(* IEC 61131-3 sources: SigmatekTestframework/src/Class/CTestScreen, 1 file *)

(* ---- CTestScreen.st ---- *)
(*!
<Class
	Name               = "CTestScreen"
	Revision           = "1.0"
	RealtimeTask       = "false"
	CyclicTask         = "false"
	BackgroundTask     = "false"
	Sigmatek           = "false"
	OSInterface        = "false"
	HighPriority       = "false"
	Automatic          = "false"
	UpdateMode         = "Prescan"
	IconPath           = ".\Class\CTestScreen\TestIcon36x36.ico"
	SharedCommandTable = "true"
	Objectsize         = "(450,120)"
	Comment            = "Base Class for Lasal Screen Testing">
	<Channels>
		<Client Name="Lse" Required="true" Internal="false" Comment="Connect to _LSE Runtime"/>
		<Client Name="m_Screen" Required="true" Internal="true"/>
		<Client Name="No" Required="true" Internal="false" Comment="Number of Screen from Lasal Screen Project"/>
	</Channels>
	<Network Name="CTestScreen">
		<!-- List of Components in this network -->
		<Components>
			<Object
				Name       = "_base"
				Class      = "CTestBase"
				Position   = "(218,120)"
				Visualized = "true">
				<Channels>
					<Server Name="Deactivate"/>
					<Server Name="State"/>
					<Client Name="cLib"/>
					<Client Name="TestSuite"/>
				</Channels>
			</Object>
			<Object
				Name       = "m_Screen"
				Class      = "CScreenInterface"
				Position   = "(210,480)"
				Visualized = "true"
				Remotely   = "true">
				<Channels>
					<Server Name="Active"/>
					<Server Name="Screen"/>
					<Client Name="ImA" Value="IMA_PICTURE"/>
					<Client Name="Lse"/>
					<Client Name="No"/>
				</Channels>
			</Object>
		</Components>
		<Comments>
		</Comments>
		<!-- List of Connections in this network -->
		<Connections>
			<Connection Source="this.State" Destination="_base.State" Vertices="(878,210),(684,210),"/>
			<Connection Source="this.Deactivate" Destination="_base.Deactivate" Vertices="(878,270),(684,270),"/>
			<Connection Source="_base.TestSuite" Destination="this.TestSuite" Vertices="(218,210),(38,210),"/>
			<Connection Source="this.m_Screen" Destination="m_Screen.Screen"/>
			<Connection Source="m_Screen.Lse" Destination="this.Lse" Vertices="(210,570),(38,330),"/>
			<Connection Source="m_Screen.No" Destination="this.No" Vertices="(210,630),(38,390),"/>
		</Connections>
		<!-- Headerfiles -->
		<Options>
		</Options>
	</Network>
</Class>
*)
#pragma using CTestBase

CTestScreen : CLASS
: CTestBase
  //Servers:
  //Clients:
	Lse 	: CltChCmd__Lse;
	No 	: CltCh_UDINT;
	m_Screen 	: CltChCmd_CScreenInterface;
  //Variables:
		m_udStartTime 	: UDINT;
		m_bTrigger 	: BOOL;
  //Functions:

	FUNCTION VIRTUAL prepare
		VAR_OUTPUT
			bRetcode 	: BOOL;
		END_VAR;

	FUNCTION VIRTUAL execute
		VAR_OUTPUT
			bRetcode 	: BOOL;
		END_VAR;

	FUNCTION VIRTUAL cleanUp
		VAR_OUTPUT
			bRetcode 	: BOOL;
		END_VAR;

	FUNCTION open
		VAR_OUTPUT
			bRetcode 	: BOOL;
		END_VAR;

	FUNCTION isActive
		VAR_OUTPUT
			bRetcode 	: BOOL;
		END_VAR;
  //Tables:
	FUNCTION @STD
		VAR_OUTPUT
			ret_code	: CONFSTATES;
		END_VAR;
	FUNCTION GLOBAL TAB @CT_;
END_CLASS;

#pragma using CScreenInterface
#pragma usingLtd _Lse

//Exclude-SccX
(*
 **********************************************************************
 * \file CTestScreen.st
 *
 * Baseclass for Testcases
 * Long description of the file.
 *
 * Copyright (c) 2016,Hoox.Software, Helmbrechts
 * All Rights Reserved.
 *
 * Created on: 01.06.2016
 *     Author: dressel
 *
 **********************************************************************
 *)

//*********************************************************************
//
//
//
//
//*********************************************************************
FUNCTION CTestScreen::open
	VAR_OUTPUT
		bRetcode 	: BOOL;
	END_VAR

   bRetcode := InsertCmd(CMD_NEWPICTURE, No$DINT, 0);

END_FUNCTION

//*********************************************************************
//
//
//
//
//*********************************************************************
FUNCTION VIRTUAL CTestScreen::prepare
	VAR_OUTPUT
		bRetcode 	: BOOL;
	END_VAR

   bRetcode := true;

END_FUNCTION
//*********************************************************************
//
//
//
//
//*********************************************************************
FUNCTION VIRTUAL CTestScreen::execute
	VAR_OUTPUT
		bRetcode 	: BOOL;
	END_VAR

   State := eStateFailed;

   bRetcode := true;

END_FUNCTION

//*********************************************************************
//
//
//
//
//*********************************************************************
FUNCTION VIRTUAL CTestScreen::cleanUp
	VAR_OUTPUT
		bRetcode 	: BOOL;
	END_VAR

   bRetcode       := true;

END_FUNCTION

//*********************************************************************
//
//
//
//
//*********************************************************************
FUNCTION CTestScreen::isActive
	VAR_OUTPUT
		bRetcode 	: BOOL;
	END_VAR

   bRetcode := (m_Screen.Active.Read() = 1);

END_FUNCTION
